RoboDK station: pickandplace.rdk

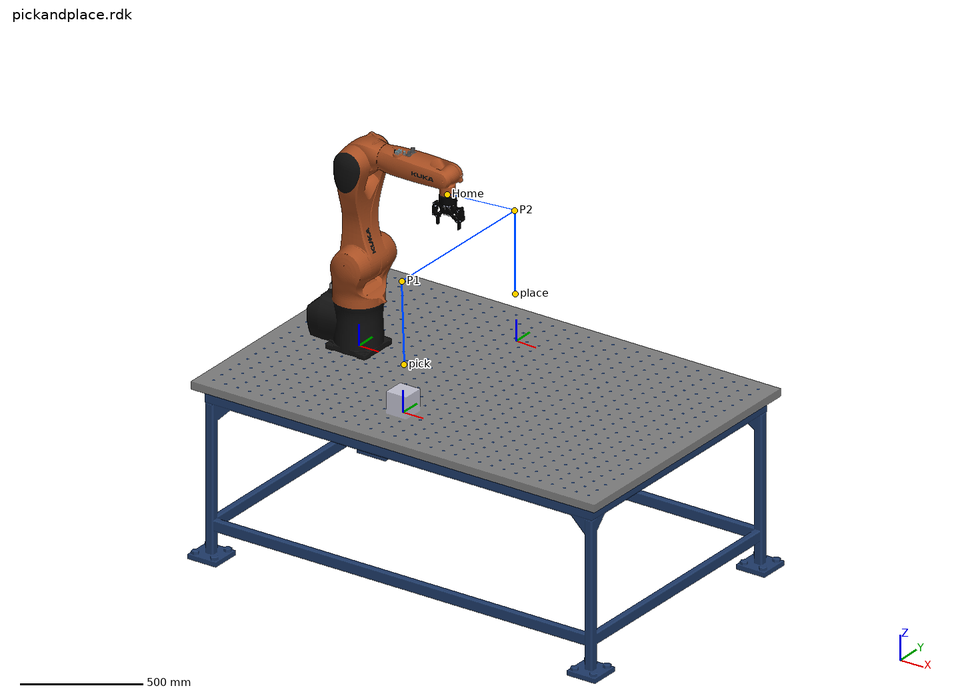
[picture v0: the station drawn from its stored meshes, robots at their saved joint values, targets as dots, program paths as lines]
Station Pick&PLace (saved by RoboDK 5.8.0). Poses are relative to the parent item; angles as X-Y-Z fixed-axis rotations.
  - frame KUKA KR 10 R900 sixx Base at (0, 0, 0) mm
    - robot KUKA KR 10 R900 sixx: 6 axes, payload 10 kg, reach 901 mm, repeatability 0.03 mm, weight 52 kg
        modified DH rows (alpha deg, a mm, theta deg, d mm): 0, 0, 0, 400; -90, 25, 0, 0; 0, 455, -90, 0; -90, 35, 0, 420; 90, 0, 0, 0; -90, 0, 180, 80
        joint limits [-170, -190, -120, -185, -120, -350] to [170, 45, 156, 185, 120, 350]; home [0, -90, 90, 0, 0, 0]; saved at [0, -90.864, 91.253, 0, 87.908, 0]
      - tool RobotiQ 2F-85 Gripper (Open), TCP at (0, 0, 0) mm, size 147.4 x 75 x 146.8 mm
  - object Table 2000x1200x800mm at (0, 0, 0) mm, size 2020 x 1340 x 800 mm, geometry from Table-2000x1200x800mm.sld
  - frame Pick at (500, -400, 0) mm
    - target Home (Cartesian target) at (-59.26, 400, 807.13) mm, rotated rx 180 ry 1.7 rz -180 deg; joints [0, -90.864, 91.253, 0, 87.908, 0] of KUKA KR 10 R900 sixx
    - target P1 (Cartesian target) at (-7.39, 2.05, 588.42) mm, rotated rx 180 ry 1.7 rz -180 deg; joints [39.068, -62.843, 86.499, -1.184, 65.027, 39.555] of KUKA KR 10 R900 sixx
    - target P2 (Cartesian target) at (-7.39, 800.9, 588.42) mm, rotated rx 180 ry 1.7 rz -180 deg; joints [-39.275, -62.619, 86.158, 1.188, 65.148, -39.762] of KUKA KR 10 R900 sixx
    - target pick (Cartesian target) at (3.73, 2.05, 214.46) mm, rotated rx 180 ry 1.7 rz -180 deg; joints [38.441, -32.735, 94.041, -2.302, 27.379, 40.473] of KUKA KR 10 R900 sixx
    - target place (Cartesian target) at (-4.19, 799.79, 214.24) mm, rotated rx -180 ry 0.35 rz -180 deg; joints [-38.908, -32.962, 94.689, 0.474, 27.998, -39.327] of KUKA KR 10 R900 sixx
    - object box at (0, 0, 50) mm, size 100 x 100 x 100 mm, geometry from box.sld
  - frame Place at (500, 400, 0) mm
  - program reset (1 instructions, listed below)
  - program main (12 instructions, listed below)
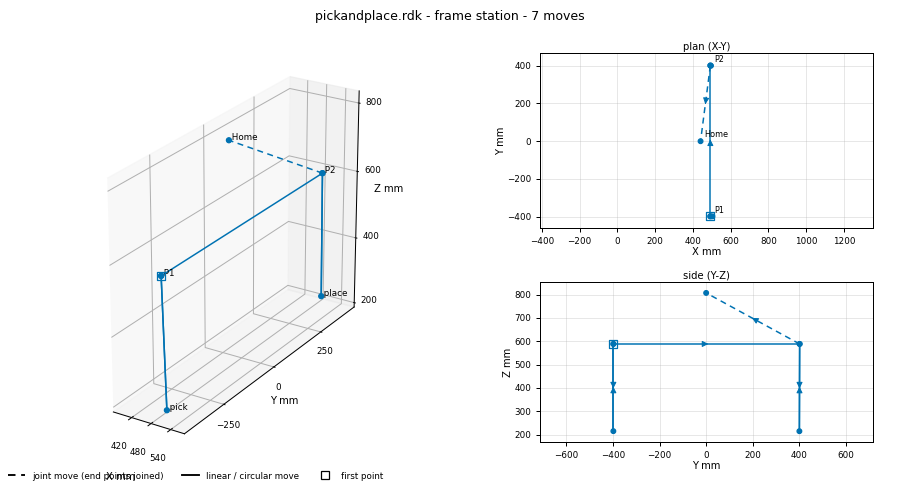
[picture p0: tool path of pickandplace.rdk in frame station, 7 of 7 moves have a stored position in this frame; points joined in program order, loops and branches not executed]

--- program reset (robot KUKA KR 10 R900 sixx) ---
  Replace objects

--- program main (robot KUKA KR 10 R900 sixx) ---
  Set Ref.: Pick
  Set Tool: RobotiQ 2F-85 Gripper (Open)
  MoveJ (P1)
  MoveL (pick)
  Attach to RobotiQ 2F-85 Gripper (Open)
  MoveL (P1)
  MoveL (P2)
  MoveL (place)
  Detach from RobotiQ 2F-85 Gripper (Open)
  MoveL (P2)
  MoveJ (Home)
  Call reset
